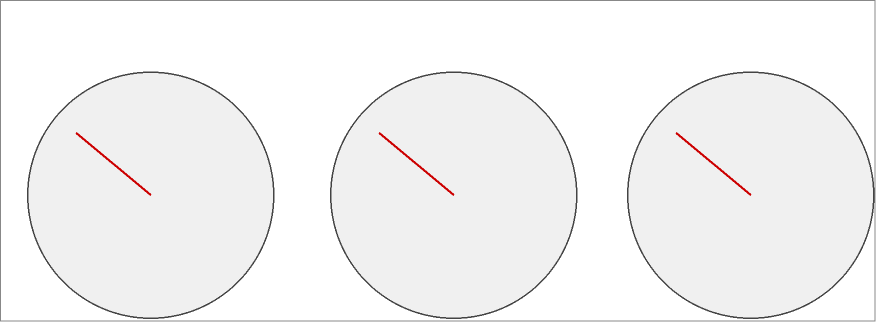
VISUALIZATION RobotinoVisu  // 876x322
    Meter360 (27,70 247x250), value: Motormesswerte.vXCartesianFromMotors, style: Meter-Meter360-Yellow, scale format: %.1f, scale -600..600
    Meter360 (330,70 247x250), value: Motormesswerte.vYCartesianFromMotors, style: Meter-Meter360-Red, scale format: %.1f, scale -600..600
    Meter360 (627,70 247x250), value: Motormesswerte.vthetaCartesianFromMotors, style: Meter-Meter360-Blue, scale format: %.1f, scale -3.1..3.41
END_VISUALIZATION

(* stored: Version 1.1.0.1, ProductVersion 3.1.4022.3
   Visu RobotinoVisu: Id {6701d034-1dde-4861-a6b5-a4770a59504d} *)
